PROGRAM MAIN
VAR
	i_xFFReset: INT;
END_VAR

(*TV1K4_VFS_01(
	i_xPMPS_OK:= TRUE, 
	i_xExt_OK:= TRUE, 
	i_xOverrideMode:= FALSE, 
	iq_stValve=> );*)

END_PROGRAM

(* stored: Version 1.1.0.1, ProductVersion 3.1.4022.18
   POU MAIN: Id {2cd28470-6329-4078-8e6a-d75c8e1492ad}, SpecialFunc None *)
